// TIA Portal V18 export
// export: Created 2026-06-08T16:04:36.8276195Z, ExportSetting WithDefaults, DisplayName Totally Integrated Automation Portal, DisplayVersion V18, DisplayName TIA Portal Openness, DisplayVersion V18, DisplayName TIA Portal Version Control Interface, DisplayVersion V18, DisplayName STEP 7 Professional, DisplayVersion V18, DisplayName STEP 7 Safety, DisplayVersion V18, DisplayName WinCC Professional, DisplayVersion V18
VAR_GLOBAL   // PLC tag table "TRUNGGIAN"
   Q_Auto_BT AT %M20.0 : Bool;   // Băng tải phân loại
   Q_Auto_Xylanh_Cao AT %M20.1 : Bool;   // Xi lanh đẩy sản phẩm cao
   Q_Auto_Xylanh_TB AT %M20.2 : Bool;   // Xi lanh đẩy sản phẩm trung bình
   Q_Manu_BT AT %M30.0 : Bool;   // Băng tải phân loại
   Q_Manu_Xylanh_Cao AT %M30.1 : Bool;   // Xi lanh đẩy sản phẩm cao
   Q_Manu_Xylanh_TB AT %M30.2 : Bool;   // Xi lanh đẩy sản phẩm trung bình
   M_Simulation AT %M5.0 : Bool;   // Nút mô phỏng trên scada
   M_Reset AT %M5.1 : Bool;   // Nút reset
   SIMU_CB_CAO AT %M5.2 : Bool;   // Mô phỏng cảm biến cao
   SIMU_CB_TB AT %M5.3 : Bool;   // Mô phỏng cảm biến trung bình
   SIMU_CB_THAP AT %M5.4 : Bool;   // Mô phỏng cảm biến thấp
END_VAR
